FUNCTION_BLOCK LogMsg
VAR_INPUT
	operationType :OperationTypeEnum ; (*Which operation to do: writing to local array or move from local to global array*)	
	Enable : BOOL;
	ptrEncoderAngle : POINTER TO REAL;
	ptrGlobalArray : POINTER TO LogGlobalArrayObj; (*Address of global array*)
	logData : LogMsgLogData; (*Log data, moved to function block, after using need to be cleared*)	
END_VAR
VAR_OUTPUT
	ErrorID : USINT;	
END_VAR
VAR_STAT
	UseFunctionSuppressBlank : BOOL := TRUE;
END_VAR

VAR

	logLocalArray : LogLocalArrayObj;
	//globalArray : REFERENCE TO LogGlobalArrayObj; (*Pointer of global array structure*)
	tempIndex : UINT;
	//encoderAngle : REFERENCE TO REAL;
	MembersToWrite	: UINT;	
	i 				: UINT;	
	NT_GetTime_0 : NT_GetTime;
	
	FB_FormatString_0:FB_FormatString;
END_VAR


CASE operationType OF
	(* Copy log message to local array *)
	COLLECT2LOCAL:
	
		IF Enable THEN (* Writing to local array only if enabled *)
			IF logLocalArray.pointers.numOfMembers < LOCAL_ARRAY_LENGTH THEN
				(* Copies data to local structure *)
				tempIndex := logLocalArray.pointers.writePointer;
				logLocalArray.array_tc[tempIndex].data := logData;
				logLocalArray.array_tc[tempIndex].TIME_TC := RTC.TimeStamp_GMT;
				//NT_GetTime_0(NETID:= ,START := TRUE,TMOUT:= ,BUSY:=,ERR:=,ERRID:= , TIMESTR=>logLocalArray.array_tc[tempIndex].TIME_TC );
				//NT_GetTime_0(START := FALSE);
				//RTC_gettime(ADR(logLocalArray.array_tc[tempIndex].TIME_TC));
				//encoderAngle ACCESS encoderAngleAddr;
				//Translates from PLC angle (0..360000) to normal angle units (0..720 degrees)
				logLocalArray.array_tc[tempIndex].Angle := REAL_TO_UINT(ptrEncoderAngle^);  //Oren// REAL_TO_UINT(floor_f((ptrEncoderAngle^*2+500)/1000.0));
				logLocalArray.pointers.writePointer := (tempIndex + 1) MOD LOCAL_ARRAY_LENGTH;
				logLocalArray.pointers.numOfMembers := logLocalArray.pointers.numOfMembers + 1;
			ELSE
				ErrorID := 1;
			END_IF;
		END_IF;	
	(* Copy all messages from local array to global array *)
	COPY2GLOBAL:

		//globalArray ACCESS globalArrayAddr;
		(*IF ptrGlobalArray^.SemData.SemID = 0 THEN
			IF globalArray.SemData.SemCreate_0.status = 0 THEN  (* SemCreate successful *)
				globalArray.SemData.SemID := globalArray.SemData.SemCreate_0.ident;  (* copy semaphore-ident the a gobal variable for global use *)
 				SemRelease(globalArray.SemData.SemID);  (* release the allocated semaphore *)
			ELSIF globalArray.SemData.SemCreate_0.status = ERR_FUB_BUSY THEN
				globalArray.SemData.SemCreate_0();
			END_IF	
		END_IF*)   

		IF	// globalArray.SemData.SemID <> 0 AND 
			//AND ptrGlobalArray^.pointers.numOfMembers < GLOBAL_ARRAY_LENGTH THEN
			logLocalArray.pointers.numOfMembers > 0 THEN
			
			IF ptrGlobalArray^.SemData.SemaStat = 0 THEN (*Allocation succesfull *)
				ptrGlobalArray^.SemData.SemaStat :=1;

				MembersToWrite := MIN(logLocalArray.pointers.numOfMembers,
										GLOBAL_ARRAY_LENGTH - ptrGlobalArray^.pointers.numOfMembers);
				MembersToWrite := MIN(MembersToWrite, MAX_MEMBERS_TO_WRITE);
				
				FOR	i := 1 TO MembersToWrite DO							
					ptrGlobalArray^.array_tc[ptrGlobalArray^.pointers.writePointer]	:= logLocalArray.array_tc[logLocalArray.pointers.readPointer];
					ptrGlobalArray^.pointers.writePointer	:= (ptrGlobalArray^.pointers.writePointer + 1)	MOD GLOBAL_ARRAY_LENGTH;
					logLocalArray.pointers.readPointer		:= (logLocalArray.pointers.readPointer + 1)		MOD LOCAL_ARRAY_LENGTH;
				END_FOR;

				logLocalArray.pointers.numOfMembers		:= logLocalArray.pointers.numOfMembers - MembersToWrite;
				ptrGlobalArray^.pointers.numOfMembers	:= ptrGlobalArray^.pointers.numOfMembers + MembersToWrite;
				
				//release semophere
				ptrGlobalArray^.SemData.SemaStat :=0;
				//SemRelease(globalArray.SemData.SemID);
				
			END_IF
		END_IF
END_CASE;

METHOD EnableLogger
VAR_INPUT
	toEnable: BOOL;
END_VAR
Enable := toEnable;
END_METHOD

METHOD FB_init : BOOL
VAR_INPUT
	bInitRetains : BOOL; // if TRUE, the retain variables are initialized (warm start / cold start)
	bInCopyCode : BOOL;  // if TRUE, the instance afterwards gets moved into the copy code (online change)
END_VAR

// beware of overriding initialization has been done by particular user
IF (ptrGlobalArray = 0) THEN
	InitLogger('LogName', 0,0);
	EnableLogger(TRUE);
END_IF
END_METHOD

//
// if globalArrayAddr and/or encoderAngleAddr is set to 0,
// so if InitLogger is called the first time, init it to defaults,
// otherwise, keep values as have been already set. 

METHOD InitLogger : BOOL
VAR_INPUT
	categoryName		: STRING[LOG_MSG_CATEGORY_LENGTH];
	globalArrayAddr		: POINTER TO LogGlobalArrayObj;
	encoderAngleAddr	: POINTER TO REAL;	
END_VAR
	THIS^.logData.category := categoryName;
	
	// if globalArrayAddr and/or encoderAngleAddr is set to 0,
	// so IF InitLogger is called the first time, init it TO defaults,
	// otherwise, keep values as have been already set. 

	IF(globalArrayAddr <> 0) THEN
		THIS^.ptrGlobalArray := globalArrayAddr;
	ELSIF(THIS^.ptrGlobalArray = 0) THEN
		THIS^.ptrGlobalArray := ADR(PcComm.LogGlobalArray);
	END_IF
	
	IF (encoderAngleAddr <> 0)THEN
		THIS^.ptrEncoderAngle := encoderAngleAddr;
	ELSIF (THIS^.ptrEncoderAngle = 0) THEN
		THIS^.ptrEncoderAngle := ADR(CONST_ZERO);
	END_IF

	InitLogger := TRUE;
END_METHOD

METHOD PUBLIC LogMsg : BOOL
VAR_INPUT
		messageLevel : enumLogMessageLevelSeverity;
		textMessage : REFERENCE TO STRING[LOG_MSG_TEXT_LENGTH];
		param1 : DINT;
		param2 : DINT;
		param3 : DINT;
		param4 : DINT;
		param5 : DINT;
		param6 : DINT;
END_VAR
	(* Copying data before putting it into local array *)
	THIS^.logData.levelSeverity := messageLevel;
	THIS^.logData.text := textMessage;
    IF (UseFunctionSuppressBlank=TRUE) THEN
        fnSuppressBlank(ADR(THIS^.logData.text));
    END_IF;
	THIS^.logData.params_tc[0] := param1;
	THIS^.logData.params_tc[1] := param2;
	THIS^.logData.params_tc[2] := param3;
	THIS^.logData.params_tc[3] := param4;
	THIS^.logData.params_tc[4] := param5;
	THIS^.logData.params_tc[5] := param6;
	THIS^.operationType := COLLECT2LOCAL;
	THIS^.logData.noParams := FALSE;	
	THIS^();
	LogMsg := TRUE;
END_METHOD

METHOD LogMsg_v2 : BOOL
VAR_INPUT
		messageLevel : enumLogMessageLevelSeverity;
		textMessage : REFERENCE TO STRING[LOG_MSG_TEXT_LENGTH];
		param1 : T_Arg;
		param2 : T_Arg;
		param3 : T_Arg;
		param4 : T_Arg;
		param5 : T_Arg;
		param6 : T_Arg;
		param7 : T_Arg;
		param8 : T_Arg;
		param9 : T_Arg;
		param10 : T_Arg;		
END_VAR
	(* Copying data before putting it into local array *)
	
	FB_FormatString_0(sFormat := textMessage,arg1 :=param1,arg2 :=param2,arg3 :=param3,arg4 :=param4,arg5 :=param5,arg6 :=param6,arg7 :=param7,arg8 :=param8,arg9 :=param9,arg10 :=param10);
	IF FB_FormatString_0.bError = FALSE THEN
		THIS^.logData.levelSeverity := messageLevel;
		THIS^.logData.text := FB_FormatString_0.sOut;
	ELSE
		THIS^.logData.text := 'Log error, Format text error';
		THIS^.logData.levelSeverity := enumLogMessageLevelSeverity.LOG_ERROR;	
	END_IF	
    IF (UseFunctionSuppressBlank=TRUE) THEN
        fnSuppressBlank(ADR(THIS^.logData.text));
    END_IF;
	THIS^.logData.noParams := TRUE;	

	THIS^.operationType := COLLECT2LOCAL;
	THIS^();
	LogMsg_v2 := TRUE;
END_METHOD

METHOD LogTransfer : BOOL
THIS^.operationType := COPY2GLOBAL;
THIS^();
LogTransfer := TRUE;
END_METHOD

END_FUNCTION_BLOCK

(* stored: Version 1.1.0.1, ProductVersion 3.1.4024.3
   POU LogMsg: Id {769126b5-6814-0808-0d67-6ca43c9f6d4b}, SpecialFunc None
   Method EnableLogger: Id {f8531278-a0d0-05fa-27e8-1d7f721a9c35}
   Method FB_init: Id {c40e4576-4208-0479-0fc2-f1b70acc21e4}
   Method InitLogger: Id {b938c9f6-d00a-0b32-0972-ab8f78a506e9}
   Method LogMsg: Id {4d062862-9240-007b-2bb1-ad05d983bae9}
   Method LogMsg_v2: Id {d512379b-9d7e-478c-84dc-daec6b9a4cc4}
   Method LogTransfer: Id {5a06fed8-3cbb-417a-ab46-6a01cbc25890} *)
